// Test/PRG_Test
PROGRAM INTERNAL PRG_Test
VAR
	fbContextBuilder_Test	: FB_ContextBuilder_Test;
	
	fbLog			: FB_LoggerLAC(Const.sLoggerFromInstance);
	
	fbScope			: FB_ScopedContext;
	bLog			: BOOL;
	bArg1			: BOOL;
	nArg2			: INT;
	sArg3			: STRING;
	
	
END_VAR

TcUnit.RUN();

IF _TaskInfo[GETCURTASKINDEXEX()].FirstCycle THEN
	// For Remote Log4TC Server change the AMS net ID and configure a route
	PRG_TaskLog.Init('127.0.0.1.1.1');
	F_Log(E_LogLevel.eInfo, 'SPS Task gestartet.');
END_IF

fbLog.Context.AddInt('logger', 42);

IF bLog THEN
	bLog := FALSE;
	F_Log(E_LogLevel.eDebug, 'Foobar'); 
	F_LogA3(E_LogLevel.eInfo, '{0}, {1}, {2}', bArg1, nArg2, sArg3);

	fbLog.Start(level := E_LogLevel.eInfo, message := 'barbaz {bLog}');
	fbLog.AddAny(bLog);
	fbLog.Context.AddString('inmessage', 'foo');
	fbLog.End();
	

	F_LogBuilder().WithLogLevel(E_LogLevel.eInfo).WithMessage('Test 1 2 3 {bLog}').WithContext(fbLog.Context).AddArg(F_BOOL(bLog)).CreateLog();
	
END_IF

PRG_TaskLog.Call();

END_PROGRAM

// ApiTest
PROGRAM INTERNAL ApiTest
VAR
	nInt			: INT;
	sStr			: STRING;
	fFloat			: REAL;
END_VAR

// Einfaches Logging
F_LogLC(
	E_LogLevel.eInfo,
	'ApiTest',
	'Log message',
	0
);

F_LogL3(
	E_LogLevel.eInfo,
	Const.sGlobalLogger, 
	'Log Message Arg={structuredArg} Arg={1} Arg=%s', 
	F_StringEx('Arg 1'),
	F_StringEx('Arg 2'),
	F_StringEx('Arg 3')
);

F_LogA3(
	E_LogLevel.eError,
	'Log Message Arg={structuredArg} Arg={1} Arg=%s',
	nInt,
	sStr,
	fFloat
);

// Einfaches Logging mit expliziten Logger
F_LogL3(
	E_LogLevel.eInfo, 
	'mbc4Log.Test',
	'Log Message Arg={structuredArg} Arg={1} Arg=%s', 
	F_StringEx('Arg 1'),
	F_StringEx('Arg 2'),
	F_StringEx('Arg 3')
);
// Einfaches Logging mit Builder
F_LogBuilder()
	.WithLogLevel(E_LogLevel.eError)
	.WithMessage('Log Message Arg={structuredArg} Arg={1} Arg=%s')
	.AddArg(F_StringEx('42')).AddArg(F_STRINGEx('Arg 2')).AddArg(F_STRINGEx('Arg 3'))
	.WithLogger('mbc4Log.Test')
	.WithContext(F_LogContext().AddInt('id', 42))
	.CreateLog();

END_PROGRAM
